{library PRIVATE}
(*
  Private Funtcion:
  Allocates a communications instance.

  Return true if station is available for allocation. 
*)

FUNCTION _AllocateInstance : BOOL
VAR_INPUT
	Instance: 				INT;		(* Instance, a number concatenated by SationNumber (1-INSTANCE_MAX_NUMBER_OF_STATIONS) and DeviceNumber (1-INSTANCE_MAX_NUMBER_OF_DEVICES). Instance is defined as: StaionNumber*100+DeviceNumber *)
END_VAR
VAR
	StationNumber: 		INT;
	StationDevice: 		INT;
END_VAR

_AllocateInstance:=FALSE;

IF _CheckInstance(Instance) THEN
	StationNumber:=Instance/100;
	StationDevice:=Instance-StationNumber*100;

	IF  ComGVL._Instance[StationNumber, StationDevice]= INSTANCE_STATUS.INSTANCE_STATUS_FREE THEN
		ComGVL._Instance[StationNumber, StationDevice]:=INSTANCE_STATUS.INSTANCE_STATUS_READY;
		_AllocateInstance:=TRUE;
	END_IF;
END_IF;

END_FUNCTION

(* stored: Version 1.1.0.1, ProductVersion 3.1.4024.2
   POU _AllocateInstance: Id {e046efc1-6aaf-4723-8440-4e45bc2614a2}, SpecialFunc None *)
